(*
SPDX-FileCopyrightText: © 2026 Oleksandr Tiutyk <trofimich@gmail.com>
SPDX-License-Identifier: MIT
License: https://opensource.org/license/mit
*)

(*!
<summary>Reports a conversion between generic type classes that the caller does not support.</summary>
<description>
The caller detects the error; this type records the supplied diagnostic values without performing the
conversion or validation. Dynamic instances and clones belong to the current task memory manager until
cleanup. Dynamic copies are explicitly registered by Clone after construction; plain __NEW does not transfer
ownership to the task manager.
</description>
*)

{attribute 'enable_dynamic_creation'}
{attribute 'no_explicit_call' := 'do not call this function block directly'}
FUNCTION_BLOCK GenericConversionNotSupportedException EXTENDS GeneralException IMPLEMENTS IGenericConversionNotSupportedException
VAR_STAT
	//! <summary>Class name shared by all instances of this function block.</summary>
	{attribute 'hide'} 
	_ClassName : STRING := __POUNAME();
END_VAR

{attribute 'monitoring' := 'call'}
PROPERTY ClassName : REFERENCE TO STRING
GET
ClassName REF= _ClassName;
END_GET
END_PROPERTY

(*!
<summary>Creates a distinct auto-disposed copy of this concrete exception type.</summary>
<description>
Copies message, code, source and timestamps through CopyGeneralFields; any prepared inner cause remains
borrowed. The current task memory manager owns the clone until cleanup. Allocation failure is terminal.
Descendants with additional payload must override Clone to preserve their type and fields. Registers the newly
constructed instance before copying payload, outside FB_init. Registration failure releases the unregistered
instance and raises a terminal error; copy failure leaves the registered instance owned by the task manager
for cleanup. Custom overrides must follow the same ownership sequence.
</description>
*)
METHOD Clone : IObject
VAR
	exceptionClone : POINTER TO GenericConversionNotSupportedException;
END_VAR
exceptionClone := __NEW(GenericConversionNotSupportedException);

IF exceptionClone = 0 THEN
	DynamicMemoryManager.RaiseAllocationFailure();
END_IF

DynamicMemoryManager.RegisterAutoDisposedObject(autoDisposedObject := exceptionClone^);

exceptionClone^.CopyGeneralFields(sourceException := THIS^);

Clone := exceptionClone^;
END_METHOD

(*!
<summary>Provides the library namespace used in diagnostics.</summary>
<description>
Borrowed read-only reference to the compiler-initialized library namespace; no ownership transfer.
</description>
*)
{attribute 'monitoring' := 'call'}
PROPERTY NamespaceName : REFERENCE TO STRING
GET
NamespaceName REF= CurrentNamespace.Name;
END_GET
END_PROPERTY

(*!
<summary>Reports the byte size of this concrete instance.</summary>
<description>
Uses XSIZEOF on the instance. Does not include separately allocated payloads or prove that an arbitrary
address is valid.
</description>
*)
{attribute 'monitoring' := 'call'}
PROPERTY SelfSize : ULINT
GET
SelfSize := XSIZEOF(THIS^);
END_GET
END_PROPERTY

(*!
<summary>Formats the supplied failure details and propagates this exception.</summary>
<description>
Call in the owning cyclic task, not during FB_init. Captures message, source and timestamps without heap
allocation during message preparation, with zero error code and no inner cause. Input storage is not retained.
Exception clone allocation failure uses the shared terminal memory mechanism.
</description>
<param name="sourceDataType">Source generic type class.</param>
<param name="targetDataType">Requested destination generic type class.</param>
*)
METHOD Throw
VAR_INPUT
	sourceNamespaceName : STRING;
	sourceClassName : STRING;
	sourcePOUName : STRING;
	sourcePosition : STRING;
	sourceDataType : GENERIC_TYPE_CLASS;
	targetDataType : GENERIC_TYPE_CLASS;
END_VAR
VAR
	message : ERROR_MESSAGE;
END_VAR
message := WideStrings.Concat255(
	"Conversion from data type '",
	TO_WSTRING(sourceDataType),
	"' to '",
	TO_WSTRING(targetDataType),
	"' is not supported");

InternalThrow(
	sourceNamespaceName := sourceNamespaceName,
	sourceClassName := sourceClassName,
	sourcePOUName := sourcePOUName,
	sourcePosition := sourcePosition,
	message := message,
	errorCode := 0,
	innerException := 0
);
END_METHOD

END_FUNCTION_BLOCK

(* stored: Version 1.1.0.1
   POU GenericConversionNotSupportedException: Id {e44deaaf-b4cd-4663-ba2a-ae13f98e6399}, SpecialFunc None
   Property ClassName: Id {efce17e5-18d7-49cc-b942-ee38809eb1c9}
   Get Get: Id {a2856dc0-811e-49cf-901c-5dd4705d623a}
   Method Clone: Id {8cd166b3-ec3f-4eee-b711-2f722b225d6b}
   Property NamespaceName: Id {40d9f937-7af3-4e76-8fb1-b7e1db2126e1}
   Get Get: Id {ae461813-a7b3-4dd0-b312-2795b4bcb283}
   Property SelfSize: Id {56727982-a3d3-474f-9c2e-6b1887ebbb2a}
   Get Get: Id {f69cf91c-0297-49b2-8571-499bd323df47}
   Method Throw: Id {62e4f95c-658a-45fb-af2f-c1637d23caa0} *)
